Staubli VAL3: Traies.pjx

--- Traies.pjx ---
Parameters version=s7.5.3 stackSize=5000 millimeterUnit=true
Data file=Traies.dtx
Type name=TrajItem path=Disk://kernel/template/TrajItem/TrajItem.pjx

--- Traies.dtx ---
public frame fFrame = {fatherId=world[0]}
public num nIndexTool
public string sID
public num nIndexFrame
public TrajItem tData
  [0]
    TrajectoryItem tSuper
      [0]
        num distance
        num moveType
        num nTime
        num nStop
        num nTcpAction
        string comment
        bool toStop
        mdesc nom_speed = {vel=450, tmax=1000}
        InstrItem iInstr[3]
          [0]
            string sType
            string sData
          [1]
            string sType
            string sData
          [2]
            string sType
            string sData
        num nMoveId
    pointRx pPoint = {fatherId=fFrame[0]}
    num nType
    pointRx pCircle = {fatherId=fFrame[0]}
